PROGRAM Stn054_PrgCalls
VAR
END_VAR


//Turn on/off by defult based on debug progress
IF gFirstScan THEN
	
	gDebug_ComponentCalls.CallStn054_15_RedGrnRecircMainMergePrestopGrn := TRUE;
	gDebug_ComponentCalls.CallStn054_16_RedGrnRecircMerge := TRUE;
	gDebug_ComponentCalls.CallStn054_17_RedGrnRecircSpurMergePrestopRed := TRUE;
	gDebug_ComponentCalls.CallStn054_22_EvalBreakStopsGrn := TRUE;
	gDebug_ComponentCalls.CallStn054_24_EmptyPuckStorageDivertGrn := TRUE;
	gDebug_ComponentCalls.CallStn054_25_EmptyPuckStorageBreakStop1Grn := TRUE;
	gDebug_ComponentCalls.CallStn054_26_EmptyPuckStorageBreakStop2Grn := TRUE;
	gDebug_ComponentCalls.CallStn054_27_EmptyPuckStorageMainMergePrestopGrn := TRUE;
	gDebug_ComponentCalls.CallStn054_28_EmptyPuckStorageSpurMergePrestopGrn := TRUE;
	gDebug_ComponentCalls.CallStn054_29_EmptyPuckStorageMergeGrn := TRUE;
	gDebug_ComponentCalls.CallStn054_30_Stn311Divert := TRUE;
	gDebug_ComponentCalls.CallStn054_31_Stn311MergePrestop := TRUE;
	gDebug_ComponentCalls.CallStn054_32_Stn311Merge := TRUE;
	gDebug_ComponentCalls.CallStn054_40_BufferRecircEntryDivertGrn := TRUE;
	gDebug_ComponentCalls.CallStn054_41_BufferRecircMainMergePrestopGrn := TRUE;
	gDebug_ComponentCalls.CallStn054_42_BufferRecircSpurMergePrestopGrn := TRUE;
	gDebug_ComponentCalls.CallStn054_43_BufferRecircMergeGrn := TRUE;
	gDebug_ComponentCalls.CallStn054_45_CleaningRecircExitDivertGrn := TRUE;
	gDebug_ComponentCalls.CallStn054_46_CleaningRecircExitMainMergePrestopGrn := TRUE;
	gDebug_ComponentCalls.CallStn054_47_CleaningRecircExitSpurMergePrestopGrn := TRUE;
	gDebug_ComponentCalls.CallStn054_48_CleaningRecircExitMergeGrn := TRUE;
	gDebug_ComponentCalls.CallStn054_50_Stn321Divert := TRUE;
	gDebug_ComponentCalls.CallStn054_51_Stn321MainMergePrestop := TRUE;
	gDebug_ComponentCalls.CallStn054_52_Stn321Merge := TRUE;
	gDebug_ComponentCalls.CallStn054_55_Stn322Divert := TRUE;
	gDebug_ComponentCalls.CallStn054_56_Stn322MainMergePrestop := TRUE;
	gDebug_ComponentCalls.CallStn054_57_Stn322Merge := TRUE;
	gDebug_ComponentCalls.CallStn054_60_Stn331Divert := TRUE;
	gDebug_ComponentCalls.CallStn054_61_Stn331MainMergePrestop := TRUE;
	gDebug_ComponentCalls.CallStn054_62_Stn331Merge := TRUE;
	gDebug_ComponentCalls.CallStn054_65_Stn332Divert := TRUE;
	gDebug_ComponentCalls.CallStn054_66_Stn332MainMergePrestop := TRUE;
	gDebug_ComponentCalls.CallStn054_67_Stn332Merge := TRUE;
	gDebug_ComponentCalls.CallStn054_75_GradingRecircEntryDivertGrn := TRUE;
	gDebug_ComponentCalls.CallStn054_76_TestRecircExitMainMergePrestopGrn := TRUE;
	gDebug_ComponentCalls.CallStn054_77_TestRecircExitSpurMergePrestopGrn := TRUE;
	gDebug_ComponentCalls.CallStn054_78_TestRecircExitMergeGrn := TRUE;
	gDebug_ComponentCalls.CallStn054_80_Stn341Divert := TRUE;
	gDebug_ComponentCalls.CallStn054_81_Stn341MainMergePrestop := TRUE;
	gDebug_ComponentCalls.CallStn054_82_Stn341Merge := TRUE;
	gDebug_ComponentCalls.CallStn054_88_Stn351Divert := TRUE;
	gDebug_ComponentCalls.CallStn054_89_Stn351MainMergePrestop := TRUE;
	gDebug_ComponentCalls.CallStn054_90_Stn351Merge := TRUE;
	gDebug_ComponentCalls.CallStn054_91_Stn352Divert := TRUE;
	gDebug_ComponentCalls.CallStn054_92_Stn352MainMergePrestop := TRUE;
	gDebug_ComponentCalls.CallStn054_93_Stn352Merge := TRUE;
	gDebug_ComponentCalls.CallStn054_95_TestRecircEntryDivertGrn := TRUE;
	gDebug_ComponentCalls.CallStn054_96_EvalRecircBreakStopsGrn := TRUE;
	
END_IF


// Conditionally Call Components
IF gDebug_ComponentCalls.CallStn054_15_RedGrnRecircMainMergePrestopGrn OR
		gFirstScan THEN
	Stn054_15_RedGrnRecircMainMergePrestopGrn();
END_IF
IF gDebug_ComponentCalls.CallStn054_16_RedGrnRecircMerge OR
		gFirstScan THEN
	Stn054_16_RedGrnRecircMerge();
END_IF
IF gDebug_ComponentCalls.CallStn054_17_RedGrnRecircSpurMergePrestopRed OR
		gFirstScan THEN
	Stn054_17_RedGrnRecircSpurMergePrestopRed();
END_IF
IF gDebug_ComponentCalls.CallStn054_22_EvalBreakStopsGrn OR
		gFirstScan THEN
	Stn054_22_EvalBreakStopsGrn();
END_IF
IF gDebug_ComponentCalls.CallStn054_24_EmptyPuckStorageDivertGrn OR
		gFirstScan THEN
	Stn054_24_EmptyPuckStorageDivertGrn();
END_IF
IF gDebug_ComponentCalls.CallStn054_25_EmptyPuckStorageBreakStop1Grn OR
		gFirstScan THEN
	Stn054_25_EmptyPuckStorageBreakStop1Grn();
END_IF
IF gDebug_ComponentCalls.CallStn054_26_EmptyPuckStorageBreakStop2Grn OR
		gFirstScan THEN
	Stn054_26_EmptyPuckStorageBreakStop2Grn();
END_IF
IF gDebug_ComponentCalls.CallStn054_27_EmptyPuckStorageMainMergePrestopGrn OR
		gFirstScan THEN
	Stn054_27_EmptyPuckStorageMainMergePrestopGrn();
END_IF
IF gDebug_ComponentCalls.CallStn054_28_EmptyPuckStorageSpurMergePrestopGrn OR
		gFirstScan THEN
	Stn054_28_EmptyPuckStorageSpurMergePrestopGrn();
END_IF
IF gDebug_ComponentCalls.CallStn054_29_EmptyPuckStorageMergeGrn OR
		gFirstScan THEN
	Stn054_29_EmptyPuckStorageMergeGrn();
END_IF
IF gDebug_ComponentCalls.CallStn054_30_Stn311Divert OR
		gFirstScan THEN
	Stn054_30_Stn311Divert();
END_IF
IF gDebug_ComponentCalls.CallStn054_31_Stn311MergePrestop OR
		gFirstScan THEN
	Stn054_31_Stn311MergePrestop();
END_IF
IF gDebug_ComponentCalls.CallStn054_32_Stn311Merge OR
		gFirstScan THEN
	Stn054_32_Stn311Merge();
END_IF
IF gDebug_ComponentCalls.CallStn054_40_BufferRecircEntryDivertGrn OR
		gFirstScan THEN
	Stn054_40_BufferRecircEntryDivertGrn();
END_IF
IF gDebug_ComponentCalls.CallStn054_41_BufferRecircMainMergePrestopGrn OR
		gFirstScan THEN
	Stn054_41_BufferRecircMainMergePrestopGrn();
END_IF
IF gDebug_ComponentCalls.CallStn054_42_BufferRecircSpurMergePrestopGrn OR
		gFirstScan THEN
	Stn054_42_BufferRecircSpurMergePrestopGrn();
END_IF
IF gDebug_ComponentCalls.CallStn054_43_BufferRecircMergeGrn OR
		gFirstScan THEN
	Stn054_43_BufferRecircMergeGrn();
END_IF
IF gDebug_ComponentCalls.CallStn054_45_CleaningRecircExitDivertGrn OR
		gFirstScan THEN
	Stn054_45_CleaningRecircExitDivertGrn();
END_IF
IF gDebug_ComponentCalls.CallStn054_46_CleaningRecircExitMainMergePrestopGrn OR
		gFirstScan THEN
	Stn054_46_CleaningRecircExitMainMergePrestopGrn();
END_IF
IF gDebug_ComponentCalls.CallStn054_47_CleaningRecircExitSpurMergePrestopGrn OR
		gFirstScan THEN
	Stn054_47_CleaningRecircExitSpurMergePrestopGrn();
END_IF
IF gDebug_ComponentCalls.CallStn054_48_CleaningRecircExitMergeGrn OR
		gFirstScan THEN
	Stn054_48_CleaningRecircExitMergeGrn();
END_IF
IF gDebug_ComponentCalls.CallStn054_50_Stn321Divert OR
		gFirstScan THEN
	Stn054_50_Stn321Divert();
END_IF
IF gDebug_ComponentCalls.CallStn054_51_Stn321MainMergePrestop OR
		gFirstScan THEN
	Stn054_51_Stn321MainMergePrestop();
END_IF
IF gDebug_ComponentCalls.CallStn054_52_Stn321Merge OR
		gFirstScan THEN
	Stn054_52_Stn321Merge();
END_IF
IF gDebug_ComponentCalls.CallStn054_55_Stn322Divert OR
		gFirstScan THEN
	Stn054_55_Stn322Divert();
END_IF
IF gDebug_ComponentCalls.CallStn054_56_Stn322MainMergePrestop OR
		gFirstScan THEN
	Stn054_56_Stn322MainMergePrestop();
END_IF
IF gDebug_ComponentCalls.CallStn054_57_Stn322Merge OR
		gFirstScan THEN
	Stn054_57_Stn322Merge();
END_IF
IF gDebug_ComponentCalls.CallStn054_60_Stn331Divert OR
		gFirstScan THEN
	Stn054_60_Stn331Divert();
END_IF
IF gDebug_ComponentCalls.CallStn054_61_Stn331MainMergePrestop OR
		gFirstScan THEN
	Stn054_61_Stn331MainMergePrestop();
END_IF
IF gDebug_ComponentCalls.CallStn054_62_Stn331Merge OR
		gFirstScan THEN
	Stn054_62_Stn331Merge();
END_IF
IF gDebug_ComponentCalls.CallStn054_65_Stn332Divert OR
		gFirstScan THEN
	Stn054_65_Stn332Divert();
END_IF
IF gDebug_ComponentCalls.CallStn054_66_Stn332MainMergePrestop OR
		gFirstScan THEN
	Stn054_66_Stn332MainMergePrestop();
END_IF
IF gDebug_ComponentCalls.CallStn054_67_Stn332Merge OR
		gFirstScan THEN
	Stn054_67_Stn332Merge();
END_IF
IF gDebug_ComponentCalls.CallStn054_75_GradingRecircEntryDivertGrn OR
		gFirstScan THEN
	Stn054_75_GradingRecircEntryDivertGrn();
END_IF
IF gDebug_ComponentCalls.CallStn054_76_TestRecircExitMainMergePrestopGrn OR
		gFirstScan THEN
	Stn054_76_TestRecircExitMainMergePrestopGrn();
END_IF
IF gDebug_ComponentCalls.CallStn054_77_TestRecircExitSpurMergePrestopGrn OR
		gFirstScan THEN
	Stn054_77_TestRecircExitSpurMergePrestopGrn();
END_IF
IF gDebug_ComponentCalls.CallStn054_78_TestRecircExitMergeGrn OR
		gFirstScan THEN
	Stn054_78_TestRecircExitMergeGrn();
END_IF
IF gDebug_ComponentCalls.CallStn054_80_Stn341Divert OR
		gFirstScan THEN
	Stn054_80_Stn341Divert();
END_IF
IF gDebug_ComponentCalls.CallStn054_81_Stn341MainMergePrestop OR
		gFirstScan THEN
	Stn054_81_Stn341MainMergePrestop();
END_IF
IF gDebug_ComponentCalls.CallStn054_82_Stn341Merge OR
		gFirstScan THEN
	Stn054_82_Stn341Merge();
END_IF
IF gDebug_ComponentCalls.CallStn054_88_Stn351Divert OR
		gFirstScan THEN
	Stn054_88_Stn351Divert();
END_IF
IF gDebug_ComponentCalls.CallStn054_89_Stn351MainMergePrestop OR
		gFirstScan THEN
	Stn054_89_Stn351MainMergePrestop();
END_IF
IF gDebug_ComponentCalls.CallStn054_90_Stn351Merge OR
		gFirstScan THEN
	Stn054_90_Stn351Merge();
END_IF
IF gDebug_ComponentCalls.CallStn054_91_Stn352Divert OR
		gFirstScan THEN
	Stn054_91_Stn352Divert();
END_IF
IF gDebug_ComponentCalls.CallStn054_92_Stn352MainMergePrestop OR
		gFirstScan THEN
	Stn054_92_Stn352MainMergePrestop();
END_IF
IF gDebug_ComponentCalls.CallStn054_93_Stn352Merge OR
		gFirstScan THEN
	Stn054_93_Stn352Merge();
END_IF
IF gDebug_ComponentCalls.CallStn054_95_TestRecircEntryDivertGrn OR
		gFirstScan THEN
	Stn054_95_TestRecircEntryDivertGrn();
END_IF
IF gDebug_ComponentCalls.CallStn054_96_EvalRecircBreakStopsGrn OR
		gFirstScan THEN
	Stn054_96_EvalRecircBreakStopsGrn();
END_IF

END_PROGRAM

(* stored: Version 1.1.0.1, ProductVersion 3.1.4024.6
   POU Stn054_PrgCalls: Id {f25742e9-8607-485c-a3e7-84bcb0ab48b9}, SpecialFunc None *)
